FUNCTION_BLOCK QuantityValue EXTENDS SM_QuantityValue
VAR_INPUT
END_VAR
VAR_OUTPUT
END_VAR
VAR
    testVar : INT;
END_VAR

SUPER^();

// do stuff

SUPER^();

END_FUNCTION_BLOCK

(* stored: Version 1.1.0.1, ProductVersion 3.1.4018.2
   POU QuantityValue: Id {6d58ff80-1670-42e4-9c84-7aa13490a2b2}, SpecialFunc None *)
